FUNCTION_BLOCK RingBuffer_Test EXTENDS FB_TestSuite
VAR
	RingBuf: RingBuffer;
	ReadBuffer: ARRAY[0..(TcTcpUdpRT_Param.RingBufferSize-1)] OF BYTE;
	WriteBuffer: ARRAY[0..(WriteBufferSize-1)] OF BYTE;
	emptyPointer: POINTER TO BYTE;
	bytePointer: BYTE;
END_VAR
VAR CONSTANT
	WriteBufferSize: UDINT := 35000;
END_VAR

//WriteWithNoDataPointer();
//WriteWithNoDataLength();
//ReadWithNoDataPointer();
//ReadWithNoDataLength();

Write3kToBufferAndEmptyIt();
ExpectBufferToBeEmpty();
ReadFromEmptyBuffer();
Write1kBytesToBuffer();
ExpectBufferNotToEmpty();

Read2kBytesFrom1kBytesBuffer();
Write25kMoreBytesToBuffer();
ExpectBufferToNotBeFull();

Read24kMoreBytesFromBuffer();
Write8kMoreBytesToBufferAndWrapAround();
Read10kMoreBytesAndWrapAround();

WriteOverflowBuffer();
WriteFullSizeOfBuffer();
ExpectBufferToBeFull();
Write1ByteOverWrapAroundAndRead1ByteOver();

METHOD ExpectBufferNotToEmpty
IF TEST_ORDERED('ExpectBufferNotToEmpty') THEN
	AssertFalse(Condition:= RingBuf.IsBufferEmpty, Message:= 'Expected IsBufferEmpty returned TRUE when the buffer was not empty');
	TEST_FINISHED();
END_IF
END_METHOD

METHOD ExpectBufferToBeEmpty
IF TEST_ORDERED('ExpectBufferToBeEmpty') THEN
	RingBuf.EmptyBuffer();
	AssertTrue(Condition:= RingBuf.IsBufferEmpty, Message:= 'Expected IsBufferEmpty returned FALSE when the buffer was empty');
	TEST_FINISHED();
END_IF
END_METHOD

METHOD ExpectBufferToBeFull
IF TEST_ORDERED('ExpectBufferToBeFull') THEN
	AssertTRUE(Condition:= RingBuf.IsBufferFull, Message:= 'Expected IsBufferFull returned FALSE when the buffer was full');
	TEST_FINISHED();
END_IF
END_METHOD

METHOD ExpectBufferToNotBeFull
IF TEST_ORDERED('ExpectBufferToNotBeFull') THEN
	AssertFalse(Condition:= RingBuf.IsBufferFull, Message:= 'Expected IsBufferFull returned TRUE when the buffer was not full');
	TEST_FINISHED();
END_IF
END_METHOD

METHOD Read10kMoreBytesAndWrapAround
VAR
	DataSize: UDINT := 10000;
	ExpectedSize: UDINT := 9000;
	Read: UDINT;
END_VAR
IF TEST_ORDERED('Read10kMoreBytesAndWrapAround') THEN
	MEMSET(destAddr:= ADR(ReadBuffer), fillByte:= 0, n:= TcTcpUdpRT_Param.RingBufferSize);
	
	Read := RingBuf.Read(Data:= ADR(ReadBuffer), Length:= DataSize);
	AssertEquals_UDINT(Expected:= ExpectedSize, Actual:= Read, Message:= CONCAT('Read data from ring buffer returned a length of ', TO_STRING(Read)));
	AssertTrue(Condition:= ReadBuffer[0] <> 0, Message:= 'The firste element was not different from zero');
	AssertTrue(Condition:= ReadBuffer[ExpectedSize-1] <> 0, Message:= 'The 8999th element was not different from zero');
	AssertTrue(Condition:= ReadBuffer[ExpectedSize] = 0, Message:= 'The 9000th element was not zero');
	AssertTrue(Condition:= ReadBuffer[DataSize] = 0, Message:= 'The last element was not zero');
	TEST_FINISHED();
END_IF
END_METHOD

METHOD Read24kMoreBytesFromBuffer
VAR
	DataSize: UDINT := 24000;
	ExpectedSize: UDINT := 24000;
	Read: UDINT;
END_VAR
IF TEST_ORDERED('Read24kMoreBytesFromBuffer') THEN
	MEMSET(destAddr:= ADR(ReadBuffer), fillByte:= 0, n:= TcTcpUdpRT_Param.RingBufferSize);
	
	Read := RingBuf.Read(Data:= ADR(ReadBuffer), Length:= DataSize);
	AssertEquals_UDINT(Expected:= ExpectedSize, Actual:= Read, Message:= CONCAT('Read data from ring buffer returned a length of ', TO_STRING(Read)));
	AssertTrue(Condition:= ReadBuffer[0] <> 0, Message:= 'The firste element was not different from zero');
	AssertTrue(Condition:= ReadBuffer[18475] <> 0, Message:= 'A random element was not different from zero');
	AssertTrue(Condition:= ReadBuffer[DataSize-1] <> 0, Message:= 'The last element was not different from zero');
	TEST_FINISHED();
END_IF
END_METHOD

METHOD Read2kBytesFrom1kBytesBuffer
VAR
	DataSize: UDINT := 2000;
	ExpectedSize: UDINT := 1000;
	Read: UDINT;
END_VAR
IF TEST_ORDERED('Read2kBytesFrom1kBytesBuffer') THEN
	MEMSET(destAddr:= ADR(ReadBuffer), fillByte:= 0, n:= TcTcpUdpRT_Param.RingBufferSize);
	
	Read := RingBuf.Read(Data:= ADR(ReadBuffer), Length:= DataSize);
	AssertEquals_UDINT(Expected:= ExpectedSize, Actual:= Read, Message:= CONCAT('Read data from ring buffer returned a length of ', TO_STRING(Read)));
	AssertTrue(Condition:= ReadBuffer[0] <> 0, Message:= 'The firste element was not different from zero');
	AssertTrue(Condition:= ReadBuffer[ExpectedSize-1] <> 0, Message:= 'The 999th element was not different from zero');
	AssertTrue(Condition:= ReadBuffer[ExpectedSize] = 0, Message:= 'The 1000th element was not zero');
	AssertTrue(Condition:= ReadBuffer[DataSize-1] = 0, Message:= 'The last element was not zero');
	TEST_FINISHED();
END_IF
END_METHOD

METHOD ReadFromEmptyBuffer
VAR
	DataSize: UDINT := 10;
	ExpectedSize: UDINT := 0;
	Read: UDINT;
END_VAR
IF TEST_ORDERED('ReadFromEmptyBuffer') THEN
	MEMSET(destAddr:= ADR(ReadBuffer), fillByte:= 0, n:= TcTcpUdpRT_Param.RingBufferSize);
	
	Read := RingBuf.Read(Data:= ADR(ReadBuffer), Length:= DataSize);
	AssertEquals_UDINT(Expected:= ExpectedSize, Actual:= Read, Message:= CONCAT('Read data from empty ring buffer returned a length of ', TO_STRING(Read)));
	TEST_FINISHED();
END_IF
END_METHOD

METHOD ReadWithNoDataLength
IF TEST_ORDERED('ReadWithNoDataLength') THEN
	emptyPointer := ADR(bytePointer);
	RingBuf.Read(Data:= emptyPointer, Length:= 0);
	AssertTrue(Condition:= RingBuf.Error, Message:= 'Reading to ring buffer did not handle a data length of zero');
	RingBuf.ResetError();
	TEST_FINISHED();
END_IF
END_METHOD

METHOD ReadWithNoDataPointer
IF TEST_ORDERED('ReadWithNoDataPointer') THEN
	emptyPointer := 0;
	RingBuf.Read(Data:= emptyPointer, Length:= 10);
	AssertTrue(Condition:= RingBuf.Error, Message:= 'Reading to ring buffer did not handle empty data pointer');
	RingBuf.ResetError();
	TEST_FINISHED();
END_IF
END_METHOD

METHOD Write1ByteOverWrapAroundAndRead1ByteOver
VAR
	DataChar1: BYTE := 55;
	DataSize1: UDINT := TcTcpUdpRT_Param.RingBufferSize - 10;
	ExpectedSize1: UDINT := TcTcpUdpRT_Param.RingBufferSize - 10;
	
	DataChar2: BYTE := 57;
	DataSize2: UDINT := 11;
	ExpectedSize2: UDINT := 11;
	
	Written: UDINT;
	Read: UDINT;
END_VAR
IF TEST_ORDERED('Write1ByteOverWrapAroundAndRead1ByteOver') THEN
	RingBuf.EmptyBuffer();
	MEMSET(destAddr:= ADR(WriteBuffer), fillByte:= DataChar1, n:= DataSize1);
	MEMSET(destAddr:= ADR(ReadBuffer), fillByte:= 0, n:= TcTcpUdpRT_Param.RingBufferSize);
	Written := RingBuf.Write(Data:= ADR(WriteBuffer), Length:= DataSize1);
	Read := RingBuf.Read(Data:= ADR(ReadBuffer), Length:= DataSize1);
	AssertEquals_UDINT(Expected:= ExpectedSize1, Actual:= Written, Message:= 'Written data to ring buffer does not match actual');
	AssertEquals_UDINT(Expected:= ExpectedSize1, Actual:= Read, Message:= CONCAT('Read data from ring buffer returned a length of ', TO_STRING(Read)));
	
	
	MEMSET(destAddr:= ADR(WriteBuffer), fillByte:= DataChar2, n:= DataSize2);
	MEMSET(destAddr:= ADR(ReadBuffer), fillByte:= 0, n:= TcTcpUdpRT_Param.RingBufferSize);
	Written := RingBuf.Write(Data:= ADR(WriteBuffer), Length:= DataSize2);
	Read := RingBuf.Read(Data:= ADR(ReadBuffer), Length:= DataSize2);
	AssertEquals_UDINT(Expected:= ExpectedSize2, Actual:= Written, Message:= 'Written data to ring buffer does not match actual');
	AssertEquals_UDINT(Expected:= ExpectedSize2, Actual:= Read, Message:= CONCAT('Read data from ring buffer returned a length of ', TO_STRING(Read)));
	AssertEquals_BYTE(Expected:= DataChar2, Actual:= ReadBuffer[ExpectedSize2-2], Message:= 'The element before wrap around was not correct');
	AssertEquals_BYTE(Expected:= DataChar2, Actual:= ReadBuffer[ExpectedSize2-1], Message:= 'The element after wrap around was not correct');
	AssertEquals_BYTE(Expected:= 0, Actual:= ReadBuffer[ExpectedSize2], Message:= 'The element after last was not zero');
	TEST_FINISHED();
END_IF
END_METHOD

METHOD Write1kBytesToBuffer
VAR
	DataChar: BYTE := 3;
	DataSize: UDINT := 1000;
	ExpectedSize: UDINT := 1000;
	Written: UDINT;
END_VAR
IF TEST_ORDERED('Write1kBytesToBuffer') THEN
	MEMSET(destAddr:= ADR(WriteBuffer), fillByte:= DataChar, n:= DataSize);
	
	Written := RingBuf.Write(Data:= ADR(WriteBuffer), Length:= DataSize);
	AssertEquals_UDINT(Expected:= ExpectedSize, Actual:= Written, Message:= 'Written data to ring buffer does not match actual');
	TEST_FINISHED();
END_IF
END_METHOD

METHOD Write25kMoreBytesToBuffer
VAR
	DataChar: BYTE := 8;
	DataSize: UDINT := 25000;
	ExpectedSize: UDINT := 25000;
	Written: UDINT;
END_VAR
IF TEST_ORDERED('Write25kMoreBytesToBuffer') THEN
	MEMSET(destAddr:= ADR(WriteBuffer), fillByte:= DataChar, n:= DataSize);
	
	Written := RingBuf.Write(Data:= ADR(WriteBuffer), Length:= DataSize);
	AssertEquals_UDINT(Expected:= ExpectedSize, Actual:= Written, Message:= 'Written data to ring buffer does not match actual');
	TEST_FINISHED();
END_IF
END_METHOD

METHOD Write3kToBufferAndEmptyIt
VAR
	DataChar: BYTE := 69;
	DataSize: UDINT := 3000;
	ExpectedSize: UDINT := 3000;
	Written: UDINT;
END_VAR
IF TEST_ORDERED('Write3kToBufferAndEmptyIt') THEN
	MEMSET(destAddr:= ADR(WriteBuffer), fillByte:= DataChar, n:= DataSize);
	
	AssertTrue(Condition:= RingBuf.IsBufferEmpty, Message:= 'Expected IsBufferEmpty returned FALSE when the buffer was empty');
	Written := RingBuf.Write(Data:= ADR(WriteBuffer), Length:= DataSize);
	AssertEquals_UDINT(Expected:= ExpectedSize, Actual:= Written, Message:= 'Written data to ring buffer does not match actual');
	AssertFalse(Condition:= RingBuf.IsBufferEmpty, Message:= 'Expected IsBufferEmpty returned TRUE when the buffer was not empty');
	
	RingBuf.EmptyBuffer();
	AssertTrue(Condition:= RingBuf.IsBufferEmpty, Message:= 'Expected IsBufferEmpty returned FALSE when the buffer was empty');
	TEST_FINISHED();
END_IF
END_METHOD

METHOD Write8kMoreBytesToBufferAndWrapAround
VAR
	DataChar: BYTE := 16;
	DataSize: UDINT := 8000;
	ExpectedSize: UDINT := 8000;
	Written: UDINT;
END_VAR
IF TEST_ORDERED('Write8kMoreBytesToBufferAndWrapAround') THEN
	MEMSET(destAddr:= ADR(WriteBuffer), fillByte:= DataChar, n:= DataSize);
	
	Written := RingBuf.Write(Data:= ADR(WriteBuffer), Length:= DataSize);
	AssertEquals_UDINT(Expected:= ExpectedSize, Actual:= Written, Message:= 'Written data to ring buffer does not match actual');
	TEST_FINISHED();
END_IF
END_METHOD

METHOD WriteFullSizeOfBuffer
VAR
	DataChar: BYTE := 24;
	DataSize: UDINT := TcTcpUdpRT_Param.RingBufferSize-1;
	ExpectedSize: UDINT := TcTcpUdpRT_Param.RingBufferSize-1;
	Written: UDINT;
END_VAR
IF TEST_ORDERED('WriteFullSizeOfBuffer') THEN
	MEMSET(destAddr:= ADR(WriteBuffer), fillByte:= DataChar, n:= DataSize);
	
	Written := RingBuf.Write(Data:= ADR(WriteBuffer), Length:= DataSize);
	AssertEquals_UDINT(Expected:= ExpectedSize, Actual:= Written, Message:= 'Written data to ring buffer does not match actual');
	AssertTrue(Condition:= RingBuf.IsBufferFull, Message:= 'Ring buffer was not full after writing full size');
	TEST_FINISHED();
END_IF
END_METHOD

METHOD WriteOverflowBuffer
VAR
	DataChar: BYTE := 16;
	DataSize: UDINT := WriteBufferSize;
	Written: UDINT;
END_VAR
IF TEST_ORDERED('WriteOverflowBuffer') THEN
	MEMSET(destAddr:= ADR(WriteBuffer), fillByte:= DataChar, n:= DataSize);
	
	Written := RingBuf.Write(Data:= ADR(WriteBuffer), Length:= DataSize);
	AssertTrue(Condition:= RingBuf.Error, Message:= RingBuf.GetError);
	RingBuf.ResetError();
	AssertFalse(Condition:= RingBuf.Error, Message:= 'Ring buffer did not reset error after overflow');
	TEST_FINISHED();
END_IF
END_METHOD

METHOD WriteWithNoDataLength
IF TEST_ORDERED('WriteWithNoDataLength') THEN
	emptyPointer := ADR(bytePointer);
	RingBuf.Write(Data:= emptyPointer, Length:= 0);
	AssertTrue(Condition:= RingBuf.Error, Message:= 'Writing to ring buffer did not handle a data length of zero');
	RingBuf.ResetError();
	TEST_FINISHED();
END_IF
END_METHOD

METHOD WriteWithNoDataPointer
IF TEST_ORDERED('WriteWithNoDataPointer') THEN
	emptyPointer := 0;
	RingBuf.Write(Data:= emptyPointer, Length:= 10);
	AssertTrue(Condition:= RingBuf.Error, Message:= 'Writing to ring buffer did not handle empty data pointer');
	RingBuf.ResetError();
	TEST_FINISHED();
END_IF
END_METHOD

END_FUNCTION_BLOCK

(* stored: Version 1.1.0.1
   POU RingBuffer_Test: Id {98565f11-6afe-01d4-1189-4324eb2e3ddd}, SpecialFunc None
   Method ExpectBufferNotToEmpty: Id {9831089e-c19c-06b8-1314-546a4c9ab050}
   Method ExpectBufferToBeEmpty: Id {75c629cb-7df8-0a9c-00a3-204a82ec8c5e}
   Method ExpectBufferToBeFull: Id {d56b2754-49b4-0e2c-38f5-5414ae6a630c}
   Method ExpectBufferToNotBeFull: Id {71444a77-0f09-0b01-244d-8f9526864a3c}
   Method Read10kMoreBytesAndWrapAround: Id {650e0902-7144-0e07-2003-8970e3c65d9e}
   Method Read24kMoreBytesFromBuffer: Id {ee2b87e8-34bb-0fba-0a93-719ed722eb85}
   Method Read2kBytesFrom1kBytesBuffer: Id {8f7ef5ee-3b62-019c-0fcd-4bb58ff0553f}
   Method ReadFromEmptyBuffer: Id {094bc8db-bd23-0901-2107-d4e36179341f}
   Method ReadWithNoDataLength: Id {35ab7352-a1bb-0626-208d-e29731a9ebc9}
   Method ReadWithNoDataPointer: Id {c7f382af-ec7f-05d4-355f-7d2ee03e149f}
   Method Write1ByteOverWrapAroundAndRead1ByteOver: Id {123120c6-1772-0bb6-3a3d-e1a2d48a9025}
   Method Write1kBytesToBuffer: Id {14a7cb7a-7ce7-0768-06fd-7b9ea6efddf3}
   Method Write25kMoreBytesToBuffer: Id {de2f9a0b-dca5-0075-2cf3-1aeec36be4fb}
   Method Write3kToBufferAndEmptyIt: Id {d58c1aa1-d401-0c98-3bcb-d7f4481a5c70}
   Method Write8kMoreBytesToBufferAndWrapAround: Id {a4bb340d-5e00-053c-3b2f-e31da388c15e}
   Method WriteFullSizeOfBuffer: Id {865e3a3f-0bec-0c0e-2c46-d8521bc62a53}
   Method WriteOverflowBuffer: Id {f75e5afd-09cf-0567-2544-dc4c2b3f1a39}
   Method WriteWithNoDataLength: Id {811e8989-8a4c-03a5-1a54-b6ef52b52cea}
   Method WriteWithNoDataPointer: Id {8ca191e7-4302-09e1-135a-7c2a877cdbb0} *)
